// TwinCAT 3 PLC project PLC1
// ProgramVersion: 3.1.4024.12
// libraries:
//   Tc2_Standard, * (Beckhoff Automation GmbH)
//   Tc2_System, * (Beckhoff Automation GmbH)
//   Tc3_Module, * (Beckhoff Automation GmbH)
// project tree:
//   FBs/Modules/ FB_LAMP_DIMM.TcPOU, FB_LAMP_ONOFF.TcPOU
//   FBs/Room/ FB_ROOM.TcPOU
//   GVLs/ Param.TcGVL
//   ITFs/Modules/ I_Lamp.TcIO
//   ITFs/Room/ I_Room.TcIO
//   / PlcTask.TcTTO
//   POUs/ MAIN.TcPOU

CONFIGURATION PLC1
    RESOURCE PLC ON TwinCAT3
        TASK PlcTask(INTERVAL := T#10ms, PRIORITY := 20);
        PROGRAM MAIN WITH PlcTask : MAIN;
    END_RESOURCE
END_CONFIGURATION

// ---- GVLs/Param.TcGVL
{attribute 'qualified_only'}
VAR_GLOBAL CONSTANT
	INDEX_START 	: INT := 0;	
	MAX_DIMM_LAMPS 	: INT := 14;
	MAX_ONOFF_LAMPS : INT := 14;	
	MAX_LAMPS		: INT := 29;
END_VAR

// ---- ITFs/Modules/I_Lamp.TcIO
INTERFACE I_Lamp

METHOD OFF : BOOL
VAR_INPUT
END_VAR
END_METHOD

METHOD ON : BOOL
VAR_INPUT
END_VAR
END_METHOD

PROPERTY State : STRING
GET
END_GET
END_PROPERTY

END_INTERFACE

// ---- ITFs/Room/I_Room.TcIO
INTERFACE I_Room

METHOD AddLamp : BOOL
VAR_INPUT
	// Lamp interface
	iLamp : I_Lamp;
END_VAR
END_METHOD

METHOD Control : BOOL
VAR_INPUT
	// Motion Sensor for the room
	bMotionSensor : BOOL;
END_VAR
END_METHOD

METHOD RemoveLamp : BOOL
VAR_INPUT
	// Lamp interface
	iLamp : I_Lamp;
END_VAR
END_METHOD

END_INTERFACE

// ---- POUs/MAIN.TcPOU
PROGRAM MAIN
VAR
	(* Classes and Interfaces *)
	fbDimm 	: ARRAY[Param.INDEX_START..Param.MAX_DIMM_LAMPS]  	OF FB_LAMP_DIMM;
	fbOnOff	: ARRAY[Param.INDEX_START..Param.MAX_ONOFF_LAMPS]  	OF FB_LAMP_ONOFF;	
	iLamp 	: ARRAY[Param.INDEX_START..Param.MAX_LAMPS] 		OF I_Lamp;
	fbRoom : FB_ROOM;

	(* Control Bits *)
	bDayMode: BOOL;
	bSensor: BOOL;
	
	(* Program Variables *)
	nIndex: INT;
	bInit: BOOL;
	nIndexOffset: INT;
END_VAR

// Initialize the array of interfaces
IF NOT bInit THEN
	// Dimmable lamps first	
	FOR nIndex := Param.INDEX_START TO Param.MAX_DIMM_LAMPS DO
		iLamp[nIndex] := fbDimm[nIndex];
	END_FOR
	
	nIndexOffset := Param.MAX_DIMM_LAMPS + 1;
	// On/Off lamps are next
	FOR nIndex := nIndexOffset TO Param.MAX_LAMPS DO
		iLamp[nIndex] := fbOnOff[nIndex - nIndexOffset];
	END_FOR
	bInit := TRUE;
END_IF

// Operating in daytime vs nighttime
IF bDayMode THEN
	FOR nIndex := Param.INDEX_START TO Param.MAX_LAMPS BY 2 DO
		fbRoom.RemoveLamp(iLamp := iLamp[nIndex]);
	END_FOR
ELSE
	FOR nIndex := Param.INDEX_START TO Param.MAX_LAMPS DO
		fbRoom.AddLamp(iLamp := iLamp[nIndex]);
	END_FOR
END_IF

// Turn on and off the lights based on a sensor
fbRoom.Control(bMotionSensor := bSensor );

END_PROGRAM

// ---- FBs/Modules/FB_LAMP_DIMM.TcPOU
{attribute 'reflection'} 
FUNCTION_BLOCK FB_LAMP_DIMM IMPLEMENTS I_Lamp
VAR
	// Hardware control variables
	fOut : REAL;
	fInc : REAL:=0.5;
	iOutHw AT %Q*:INT;
	
	// Instance-path variable
    {attribute 'instance-path'} 
    {attribute 'noinit'} 
    sPath : STRING; 
END_VAR

METHOD OFF : BOOL
// Intensity in 0..100% variable fOut
fOut := fOut - fInc;
IF fOut < 0.0 THEN
	fOut := 0.0;
END_IF

// Conversion to hardware output 0..32767
iOutHw := LIMIT(0,REAL_TO_INT(fOut * 327.67), 32767);
END_METHOD

METHOD ON : BOOL
// Intensity in 0..100% variable fOut
fOut := fOut + fInc;
IF fOut > 100.0 THEN
	fOut := 100.0;
END_IF

// Conversion to hardware output 0..32767
iOutHw := LIMIT(0,REAL_TO_INT(fOut * 327.67), 32767);
END_METHOD

PROPERTY State : STRING
GET
State := CONCAT('Object: ', sPath);
State := CONCAT(State, ' State (%):');
State := CONCAT(State, REAL_TO_STRING(THIS^.fOut));
END_GET
END_PROPERTY

END_FUNCTION_BLOCK

// ---- FBs/Modules/FB_LAMP_ONOFF.TcPOU
{attribute 'reflection'} 
FUNCTION_BLOCK FB_LAMP_ONOFF IMPLEMENTS I_Lamp
VAR	
	// Hardware control variables
	bOutHw AT %Q*:BOOL;
	
	// Instance-path variable
    {attribute 'instance-path'} 
    {attribute 'noinit'} 
    sPath : STRING; 
END_VAR

METHOD OFF : BOOL
bOutHw := FALSE;
END_METHOD

METHOD ON : BOOL
bOutHw := TRUE;
END_METHOD

PROPERTY State : STRING
GET
State := CONCAT('Object: ', sPath);
State := CONCAT(State, ' State:');
State := CONCAT(State, BOOL_TO_STRING(THIS^.bOutHw));
END_GET
END_PROPERTY

END_FUNCTION_BLOCK

// ---- FBs/Room/FB_ROOM.TcPOU
FUNCTION_BLOCK FB_ROOM IMPLEMENTS I_Room
VAR
	// Array of registered lamps
	iLamps 		: ARRAY[Param.INDEX_START..Param.MAX_LAMPS] OF I_Lamp;
END_VAR

METHOD AddLamp : BOOL
VAR_INPUT
	(* Lamp interface*)
	iLamp	: I_Lamp;
END_VAR

VAR
	// Loop Counter
	nIndex	: INT;
END_VAR
AddLamp := FALSE;
// Check to see if the reference is valid, if not return immediately
IF (iLamp = 0) THEN
	RETURN;
END_IF

// Is the lamp already registered?
FOR nIndex := Param.INDEX_START TO Param.MAX_LAMPS DO
	IF (THIS^.iLamps[nIndex] = iLamp) THEN
		AddLamp := TRUE;
		RETURN;
	END_IF
END_FOR

// Save it to the array if it's not
FOR nIndex := Param.INDEX_START TO  Param.MAX_LAMPS DO
	IF (THIS^.iLamps[nIndex] = 0) THEN
		THIS^.iLamps[nIndex] := iLamp;
		AddLamp := TRUE;
		EXIT;					
	END_IF
END_FOR
END_METHOD

METHOD Control : BOOL
VAR_INPUT
	(* Motion Sensor for the room*)
	bMotionSensor	: BOOL;
END_VAR

VAR
	nIndex: INT;
END_VAR
Control := FALSE;
FOR nIndex := Param.INDEX_START TO  Param.MAX_LAMPS DO
	IF bMotionSensor AND (THIS^.iLamps[nIndex] <> 0) THEN
		iLamps[nIndex].ON();
		Control := TRUE;
	ELSIF (THIS^.iLamps[nIndex] <> 0) THEN
		iLamps[nIndex].OFF();
	END_IF
END_FOR
END_METHOD

METHOD FB_exit : BOOL
VAR_INPUT
	bInCopyCode : BOOL; // if TRUE, the exit method is called for exiting an instance that is copied afterwards (online change).
END_VAR

VAR
	nIndex: INT;
END_VAR
FOR nIndex := 1 TO Param.MAX_LAMPS DO
	iLamps[nIndex] := 16#00;
END_FOR
END_METHOD

METHOD RemoveLamp : BOOL
VAR_INPUT
	(* Lamp interface*)
	iLamp	: I_Lamp;
END_VAR

VAR
	// Loop Counter
	nIndex	: INT;
END_VAR
RemoveLamp := FALSE;

IF (iLamp = 0) THEN
	RETURN;
END_IF

FOR nIndex := Param.INDEX_START TO  Param.MAX_LAMPS DO
	IF (THIS^.iLamps[nIndex] = iLamp) THEN
		THIS^.iLamps[nIndex] := 0;
		RemoveLamp := TRUE;	
	END_IF
END_FOR
END_METHOD

END_FUNCTION_BLOCK
